TYPE ST_SafetyGroup :
STRUCT
    Name : STRING;
    RunGroup AT %Q* : BOOL := TRUE; //Auto default to run state
    AckGroup AT %Q* : BOOL;
    
    Diag AT %I* : BYTE;
    Status AT %I* : BYTE;
    groupState : E_SafetyGroupState;
END_STRUCT
END_TYPE

(* stored: Version 1.1.0.1, ProductVersion 3.1.4024.11
   DUT ST_SafetyGroup: Id {4a23a734-2f5d-471e-98da-543899da80e2} *)
